(* Logix 5000 project; controller PRU vendor 1 type 14 code 107 rev 20.13; software revision 20.01; part 15 of 17 *)
(* tags used below, declared in another part *)
   AFI : BOOL;
   CMD_LEFT_SCREW_START : BOOL;
   CMD_LEFT_SCREW_STOP : BOOL;
   CMD_RIGHT_SCREW_START : BOOL;
   CMD_RIGHT_SCREW_STOP : BOOL;
   CONTROLLED_STOP : BOOL;
   COOL_FOR_MOTOR_STOP : BOOL;
   DCS_ESTOP_ION : BOOL;
   DRYER : DUAL_SCREW;
   DRYER_AUTO_MODE_PB_ONS : BOOL;
   DRYER_CENTER_STARTUP_MODE : BOOL;
   DRYER_CENTER_TON : TIMER;
   DRYER_MAN_MODE_PB_ONS : BOOL;
   DRYER_MODE_AUTO : BOOL;
   DRYER_MODE_OFF : BOOL;
   DRYER_ONS : BOOL;
   DRYER_SEMIAUTO_MODE_PB_ONS : BOOL;
   DRYER_SHUTDOWN_FAULT_ION : BOOL;
   ENCODER_ERROR : REAL;
   ESR_CONTACT_1_ION : BOOL;
   ESR_CONTACT_2_ION : BOOL;
   ESTOP_PB_IOF : BOOL;   // E-STOP PUSHBUTTON IS PUSHED.
   FAULT : DINT[100];
   FAULT_DRYERL_MSG_TON : TIMER;
   FAULT_DRYERR_MSG_TON : TIMER;
   FAULT_TIMER : TIMER[10000];
   FAULTS_FA1_IOK : BOOL;   // SYSTEM LEVEL FAULTS ARE OK.
   FAULTS_FA1A_IOK : BOOL;   // MODULE FAULTS ARE OK.
   FAULTS_FA1B_IOK : BOOL;   // STOP PUSHBUTTON FAULTS ARE OK.
   FAULTS_FA3A_IOK : BOOL;   // SCREWS DRIVES NOT FAULTED.
   HMI_ALARM_RESET : BOOL;
   HMI_DRYER_AUTO_MODE_PB : BOOL;
   HMI_DRYER_MAN_MODE_PB : BOOL;
   HMI_DRYER_OFF_MODE_PB : BOOL;
   HMI_DRYER_SEMIAUTO_MODE_PB : BOOL;
   HMI_DRYERL_SPEED : REAL;
   HMI_DRYERR_SPEED : REAL;
   HMI_STOP_ALL : BOOL;
   HMI_SYSTEM_AUTO_MODE_PB : BOOL;
   HMI_VFD_1_JOG_FWD_PB : BOOL;
   HMI_VFD_1_JOG_REV_PB : BOOL;
   HMI_VFD_2_JOG_FWD_PB : BOOL;
   HMI_VFD_2_JOG_REV_PB : BOOL;
   MODE_DRYER : INT;
   Module_DRYERL_Fault : DINT;
   Module_DRYERL_Iok : BOOL;
   Module_DRYERL_Status : DINT;
   Module_DRYERR_Fault : DINT;
   Module_DRYERR_Iok : BOOL;
   Module_DRYERR_Status : DINT;
   OK_TO_STOP : BOOL;
   PF70EL_Message : MESSAGE;
   PF70ER_Message : MESSAGE;
   PROCESS_SEQUENCER : INT;
   REQUEST_TO_STOP : BOOL;   // HMI MIXING SCREEN - REQUEST TO STOP WHEN SCREWS ARE NEAR ZERO.
   REQUEST_TO_STOP_L : BOOL;
   SCREWS_ENABLE_GON : BOOL;   // Dryer screw faults are ok.
   THRESHOLD : REAL[9000];
   VFD_1_Current_Real : REAL;
   VFD_2_Current_Real : REAL;
   VFD_CommsFaultTest : DINT;
   VFDS_BON : BOOL;   // DRYER VFDs HAVE BEEN COMMANDED ON FOR 1 SECOND.
   VFDS_TON : TIMER;

PROGRAM SCREW_CONTROL   (* main routine DUALSCREW *)

ROUTINE A01_DRYER_Start_Stop   (* ladder *)
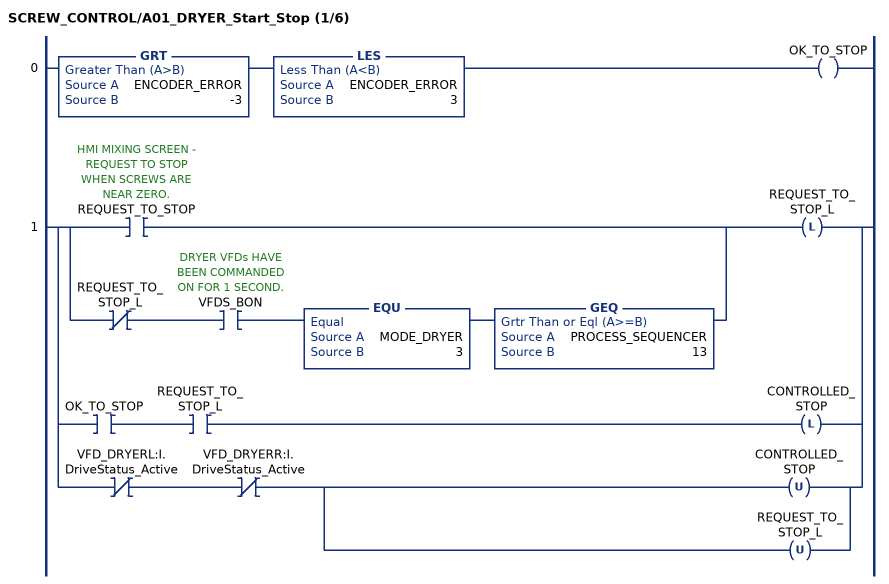
   0: GRT(ENCODER_ERROR,-3)LES(ENCODER_ERROR,3)OTE(OK_TO_STOP);
   1: [[XIC(REQUEST_TO_STOP) ,XIO(REQUEST_TO_STOP_L) XIC(VFDS_BON) EQU(MODE_DRYER,3) GEQ(PROCESS_SEQUENCER,13) ] OTL(REQUEST_TO_STOP_L) ,XIC(OK_TO_STOP) XIC(REQUEST_TO_STOP_L) OTL(CONTROLLED_STOP) ,XIO(VFD_DRYERL:I.DriveStatus_Active) XIO(VFD_DRYERR:I.DriveStatus_Active) [OTU(CONTROLLED_STOP) ,OTU(REQUEST_TO_STOP_L) ] ];
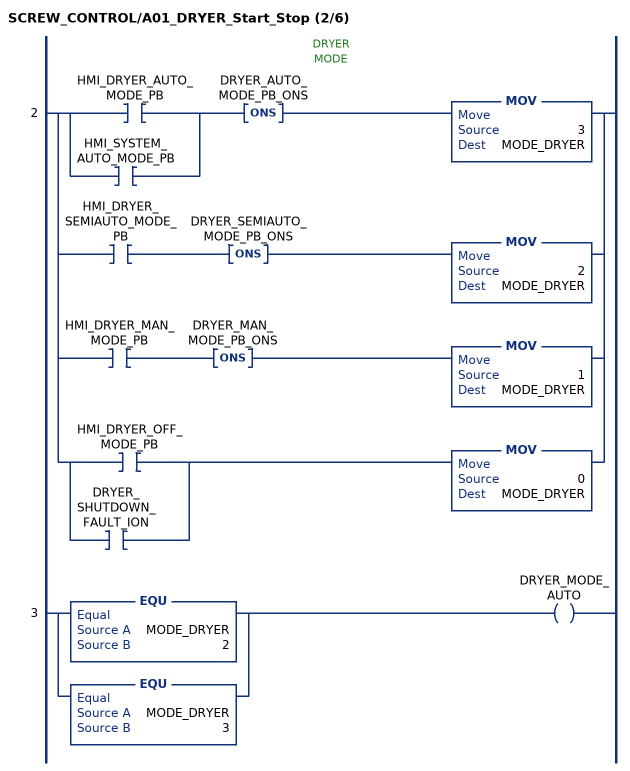
   // DRYER
   // MODE
   2: [[XIC(HMI_DRYER_AUTO_MODE_PB) ,XIC(HMI_SYSTEM_AUTO_MODE_PB) ] ONS(DRYER_AUTO_MODE_PB_ONS) MOV(3,MODE_DRYER) ,XIC(HMI_DRYER_SEMIAUTO_MODE_PB) ONS(DRYER_SEMIAUTO_MODE_PB_ONS) MOV(2,MODE_DRYER) ,XIC(HMI_DRYER_MAN_MODE_PB) ONS(DRYER_MAN_MODE_PB_ONS) MOV(1,MODE_DRYER) ,[XIC(HMI_DRYER_OFF_MODE_PB) ,XIC(DRYER_SHUTDOWN_FAULT_ION) ] MOV(0,MODE_DRYER) ];
   3: [EQU(MODE_DRYER,2) ,EQU(MODE_DRYER,3) ]OTE(DRYER_MODE_AUTO);
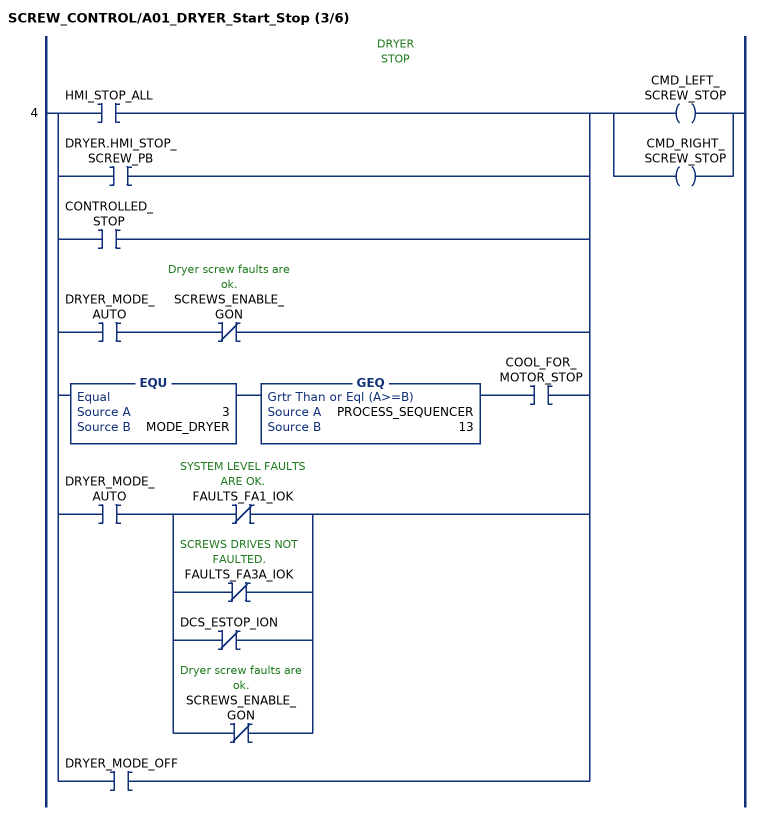
   // DRYER
   // STOP
   4: [XIC(HMI_STOP_ALL) ,XIC(DRYER.HMI_STOP_SCREW_PB) ,XIC(CONTROLLED_STOP) ,XIC(DRYER_MODE_AUTO) XIO(SCREWS_ENABLE_GON) ,EQU(3,MODE_DRYER) GEQ(PROCESS_SEQUENCER,13) XIC(COOL_FOR_MOTOR_STOP) ,XIC(DRYER_MODE_AUTO) [XIO(FAULTS_FA1_IOK) ,XIO(FAULTS_FA3A_IOK) ,XIO(DCS_ESTOP_ION) ,XIO(SCREWS_ENABLE_GON) ] ,XIC(DRYER_MODE_OFF) ][OTE(CMD_LEFT_SCREW_STOP) ,OTE(CMD_RIGHT_SCREW_STOP) ];
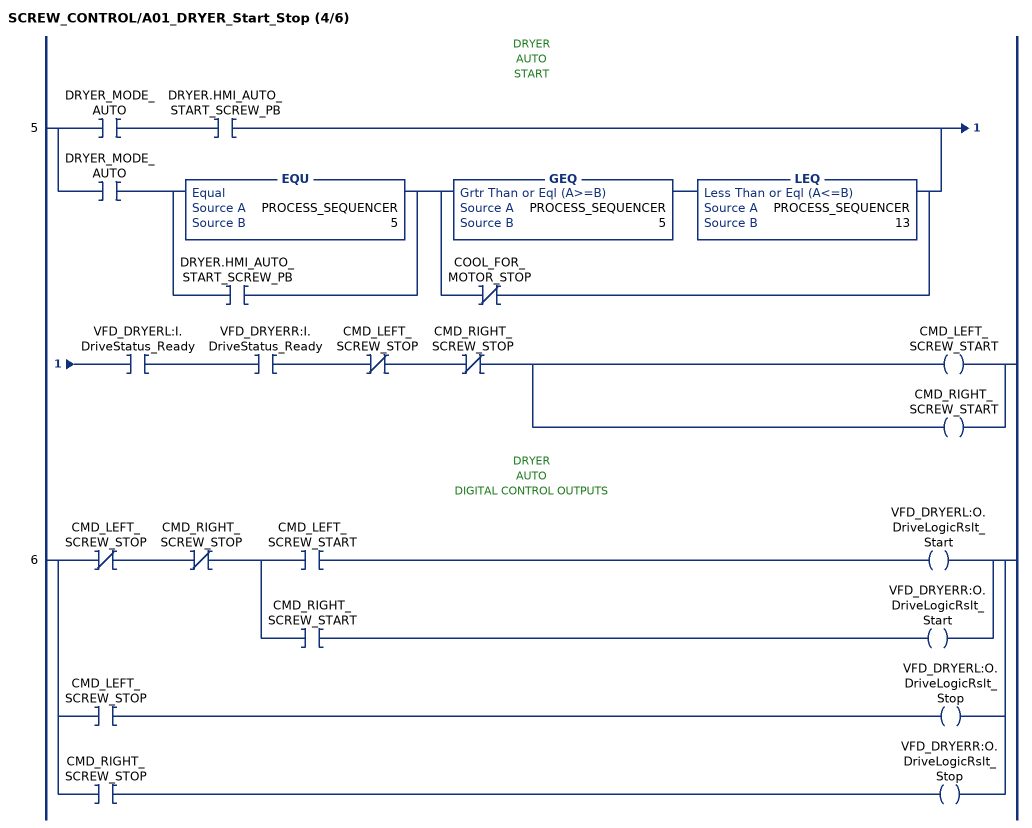
   // DRYER
   // AUTO
   //  START
   5: [XIC(DRYER_MODE_AUTO) XIC(DRYER.HMI_AUTO_START_SCREW_PB) ,XIC(DRYER_MODE_AUTO) [EQU(PROCESS_SEQUENCER,5) ,XIC(DRYER.HMI_AUTO_START_SCREW_PB) ] [GEQ(PROCESS_SEQUENCER,5) LEQ(PROCESS_SEQUENCER,13) ,XIO(COOL_FOR_MOTOR_STOP) ] ]XIC(VFD_DRYERL:I.DriveStatus_Ready)XIC(VFD_DRYERR:I.DriveStatus_Ready)XIO(CMD_LEFT_SCREW_STOP)XIO(CMD_RIGHT_SCREW_STOP)[OTE(CMD_LEFT_SCREW_START) ,OTE(CMD_RIGHT_SCREW_START) ];
   // DRYER
   // AUTO
   // DIGITAL CONTROL OUTPUTS
   6: [XIO(CMD_LEFT_SCREW_STOP) XIO(CMD_RIGHT_SCREW_STOP) [XIC(CMD_LEFT_SCREW_START) OTE(VFD_DRYERL:O.DriveLogicRslt_Start) ,XIC(CMD_RIGHT_SCREW_START) OTE(VFD_DRYERR:O.DriveLogicRslt_Start) ] ,XIC(CMD_LEFT_SCREW_STOP) OTE(VFD_DRYERL:O.DriveLogicRslt_Stop) ,XIC(CMD_RIGHT_SCREW_STOP) OTE(VFD_DRYERR:O.DriveLogicRslt_Stop) ];
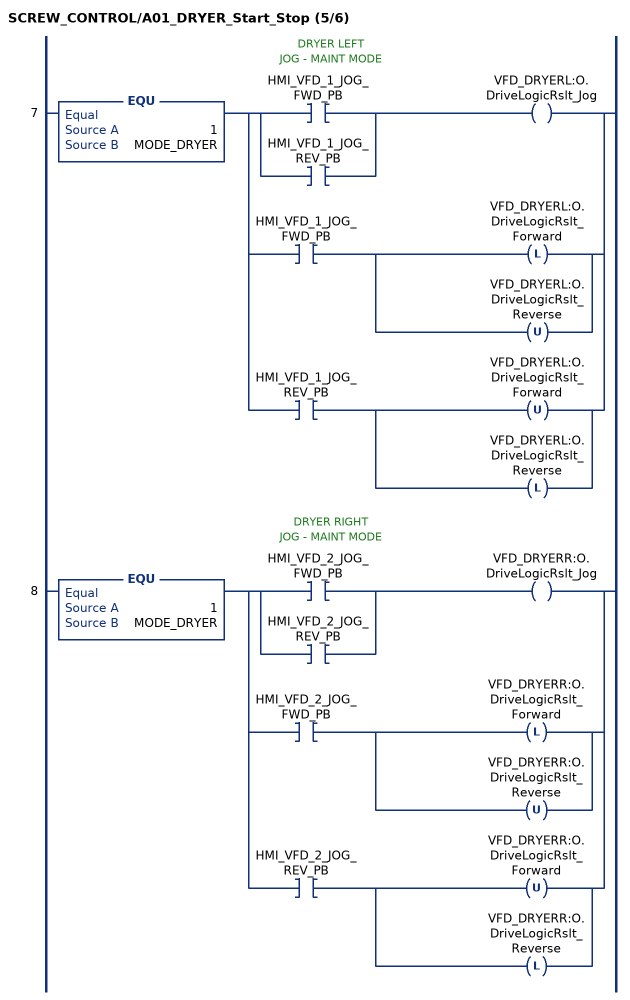
   // DRYER LEFT
   // JOG - MAINT MODE
   7: EQU(1,MODE_DRYER)[[XIC(HMI_VFD_1_JOG_FWD_PB) ,XIC(HMI_VFD_1_JOG_REV_PB) ] OTE(VFD_DRYERL:O.DriveLogicRslt_Jog) ,XIC(HMI_VFD_1_JOG_FWD_PB) [OTL(VFD_DRYERL:O.DriveLogicRslt_Forward) ,OTU(VFD_DRYERL:O.DriveLogicRslt_Reverse) ] ,XIC(HMI_VFD_1_JOG_REV_PB) [OTU(VFD_DRYERL:O.DriveLogicRslt_Forward) ,OTL(VFD_DRYERL:O.DriveLogicRslt_Reverse) ] ];
   // DRYER RIGHT
   // JOG - MAINT MODE
   8: EQU(1,MODE_DRYER)[[XIC(HMI_VFD_2_JOG_FWD_PB) ,XIC(HMI_VFD_2_JOG_REV_PB) ] OTE(VFD_DRYERR:O.DriveLogicRslt_Jog) ,XIC(HMI_VFD_2_JOG_FWD_PB) [OTL(VFD_DRYERR:O.DriveLogicRslt_Forward) ,OTU(VFD_DRYERR:O.DriveLogicRslt_Reverse) ] ,XIC(HMI_VFD_2_JOG_REV_PB) [OTU(VFD_DRYERR:O.DriveLogicRslt_Forward) ,OTL(VFD_DRYERR:O.DriveLogicRslt_Reverse) ] ];
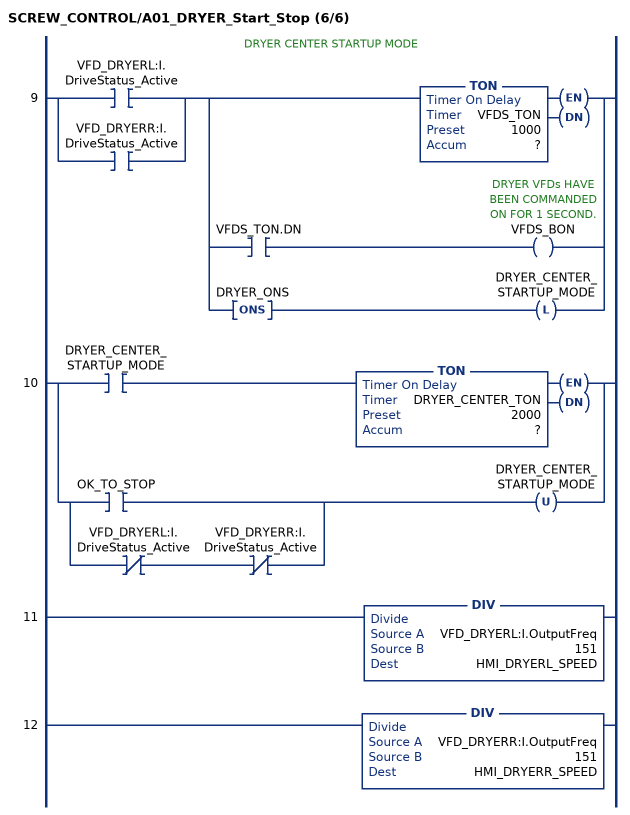
   // DRYER CENTER STARTUP MODE
   9: [XIC(VFD_DRYERL:I.DriveStatus_Active) ,XIC(VFD_DRYERR:I.DriveStatus_Active) ][TON(VFDS_TON,?,?) ,XIC(VFDS_TON.DN) OTE(VFDS_BON) ,ONS(DRYER_ONS) OTL(DRYER_CENTER_STARTUP_MODE) ];
   10: [XIC(DRYER_CENTER_STARTUP_MODE) TON(DRYER_CENTER_TON,?,?) ,[XIC(OK_TO_STOP) ,XIO(VFD_DRYERL:I.DriveStatus_Active) XIO(VFD_DRYERR:I.DriveStatus_Active) ] OTU(DRYER_CENTER_STARTUP_MODE) ];
   11: DIV(VFD_DRYERL:I.OutputFreq,151,HMI_DRYERL_SPEED);
   12: DIV(VFD_DRYERR:I.OutputFreq,151,HMI_DRYERR_SPEED);
END_ROUTINE

ROUTINE B01_FA1_B_FAULTS_1200_STOP   (* ladder *)
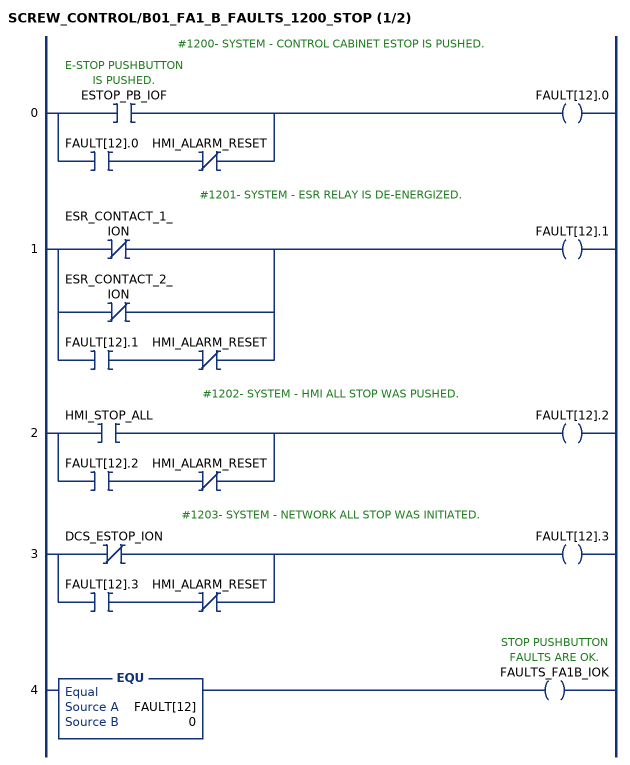
   // #1200- SYSTEM - CONTROL CABINET ESTOP IS PUSHED.
   0: [XIC(ESTOP_PB_IOF) ,XIC(FAULT[12].0) XIO(HMI_ALARM_RESET) ]OTE(FAULT[12].0);
   // #1201- SYSTEM - ESR RELAY IS DE-ENERGIZED.
   1: [XIO(ESR_CONTACT_1_ION) ,XIO(ESR_CONTACT_2_ION) ,XIC(FAULT[12].1) XIO(HMI_ALARM_RESET) ]OTE(FAULT[12].1);
   // #1202- SYSTEM - HMI ALL STOP WAS PUSHED.
   2: [XIC(HMI_STOP_ALL) ,XIC(FAULT[12].2) XIO(HMI_ALARM_RESET) ]OTE(FAULT[12].2);
   // #1203- SYSTEM - NETWORK ALL STOP WAS INITIATED.
   3: [XIO(DCS_ESTOP_ION) ,XIC(FAULT[12].3) XIO(HMI_ALARM_RESET) ]OTE(FAULT[12].3);
   4: EQU(FAULT[12],0)OTE(FAULTS_FA1B_IOK);
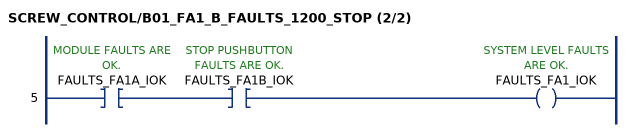
   5: XIC(FAULTS_FA1A_IOK)XIC(FAULTS_FA1B_IOK)OTE(FAULTS_FA1_IOK);
END_ROUTINE

ROUTINE B03_FA3_A_PYROSCREW_FAULTS_3000   (* ladder *)
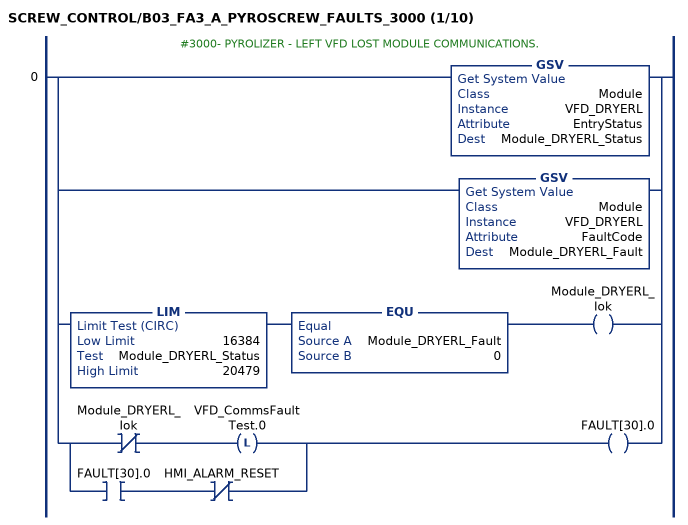
   // #3000- PYROLIZER - LEFT VFD LOST MODULE COMMUNICATIONS.
   0: [GSV(Module,VFD_DRYERL,EntryStatus,Module_DRYERL_Status) ,GSV(Module,VFD_DRYERL,FaultCode,Module_DRYERL_Fault) ,LIM(16384,Module_DRYERL_Status,20479) EQU(Module_DRYERL_Fault,0) OTE(Module_DRYERL_Iok) ,[XIO(Module_DRYERL_Iok) OTL(VFD_CommsFaultTest.0) ,XIC(FAULT[30].0) XIO(HMI_ALARM_RESET) ] OTE(FAULT[30].0) ];
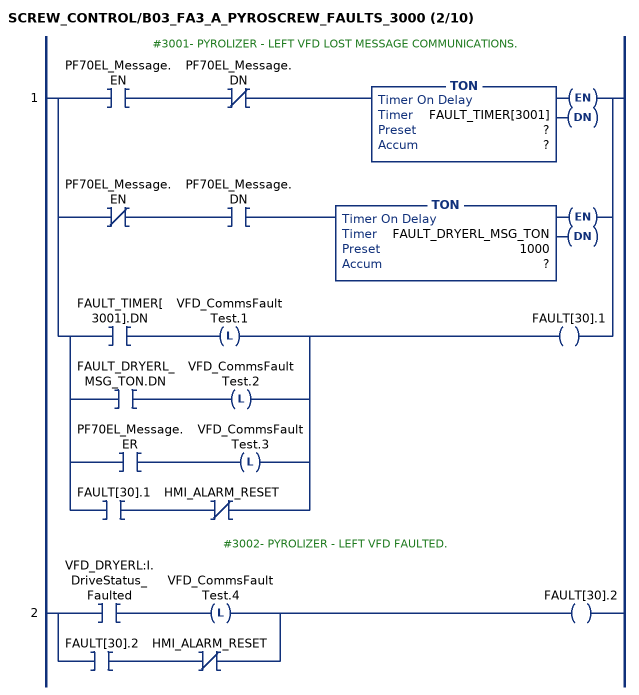
   // #3001- PYROLIZER - LEFT VFD LOST MESSAGE COMMUNICATIONS.
   1: [XIC(PF70EL_Message.EN) XIO(PF70EL_Message.DN) TON(FAULT_TIMER[3001],?,?) ,XIO(PF70EL_Message.EN) XIC(PF70EL_Message.DN) TON(FAULT_DRYERL_MSG_TON,?,?) ,[XIC(FAULT_TIMER[3001].DN) OTL(VFD_CommsFaultTest.1) ,XIC(FAULT_DRYERL_MSG_TON.DN) OTL(VFD_CommsFaultTest.2) ,XIC(PF70EL_Message.ER) OTL(VFD_CommsFaultTest.3) ,XIC(FAULT[30].1) XIO(HMI_ALARM_RESET) ] OTE(FAULT[30].1) ];
   // #3002- PYROLIZER - LEFT VFD FAULTED.
   2: [XIC(VFD_DRYERL:I.DriveStatus_Faulted) OTL(VFD_CommsFaultTest.4) ,XIC(FAULT[30].2) XIO(HMI_ALARM_RESET) ]OTE(FAULT[30].2);
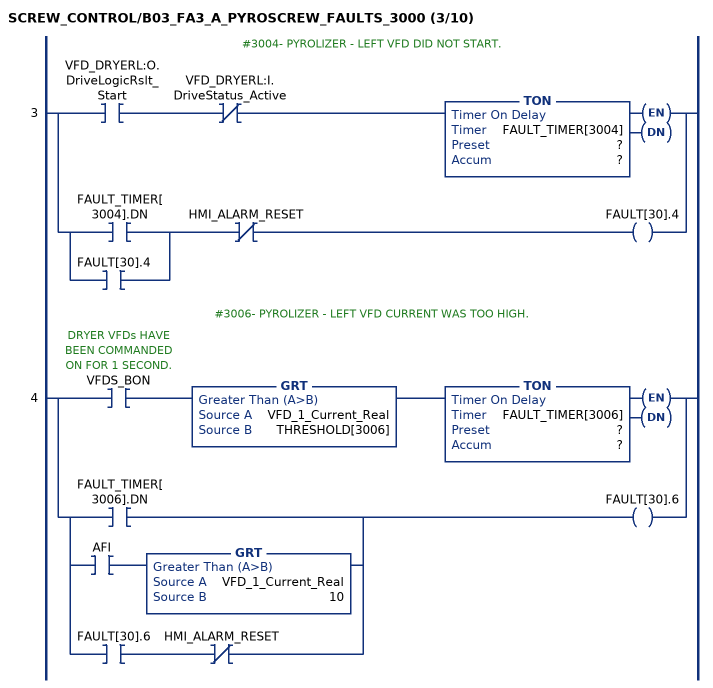
   // #3004- PYROLIZER - LEFT VFD DID NOT START.
   3: [XIC(VFD_DRYERL:O.DriveLogicRslt_Start) XIO(VFD_DRYERL:I.DriveStatus_Active) TON(FAULT_TIMER[3004],?,?) ,[XIC(FAULT_TIMER[3004].DN) ,XIC(FAULT[30].4) ] XIO(HMI_ALARM_RESET) OTE(FAULT[30].4) ];
   // #3006- PYROLIZER - LEFT VFD CURRENT WAS TOO HIGH.
   4: [XIC(VFDS_BON) GRT(VFD_1_Current_Real,THRESHOLD[3006]) TON(FAULT_TIMER[3006],?,?) ,[XIC(FAULT_TIMER[3006].DN) ,XIC(AFI) GRT(VFD_1_Current_Real,10) ,XIC(FAULT[30].6) XIO(HMI_ALARM_RESET) ] OTE(FAULT[30].6) ];
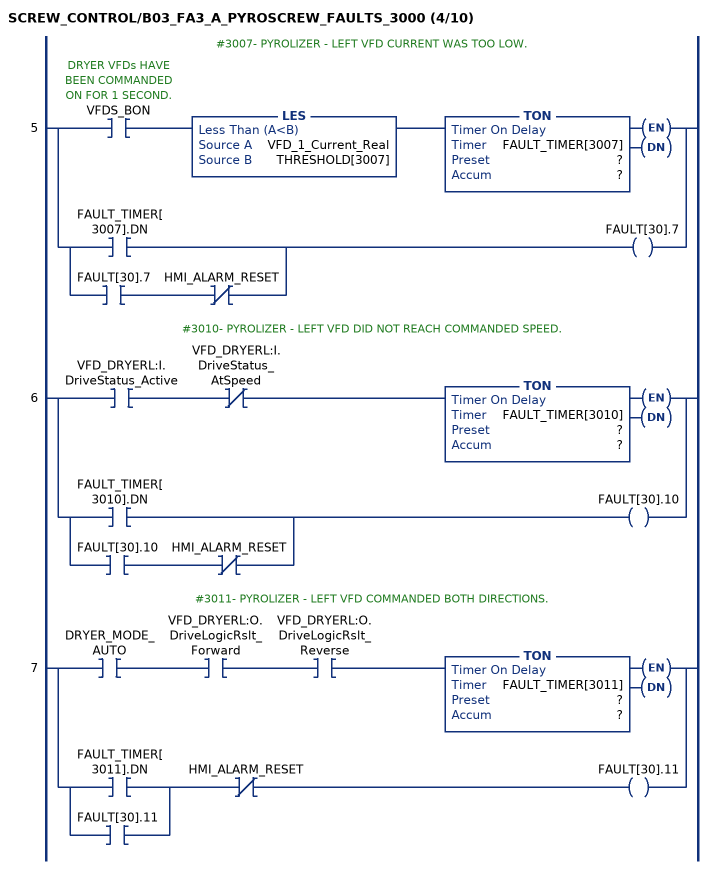
   // #3007- PYROLIZER - LEFT VFD CURRENT WAS TOO LOW.
   5: [XIC(VFDS_BON) LES(VFD_1_Current_Real,THRESHOLD[3007]) TON(FAULT_TIMER[3007],?,?) ,[XIC(FAULT_TIMER[3007].DN) ,XIC(FAULT[30].7) XIO(HMI_ALARM_RESET) ] OTE(FAULT[30].7) ];
   // #3010- PYROLIZER - LEFT VFD DID NOT REACH COMMANDED SPEED.
   6: [XIC(VFD_DRYERL:I.DriveStatus_Active) XIO(VFD_DRYERL:I.DriveStatus_AtSpeed) TON(FAULT_TIMER[3010],?,?) ,[XIC(FAULT_TIMER[3010].DN) ,XIC(FAULT[30].10) XIO(HMI_ALARM_RESET) ] OTE(FAULT[30].10) ];
   // #3011- PYROLIZER - LEFT VFD COMMANDED BOTH DIRECTIONS.
   7: [XIC(DRYER_MODE_AUTO) XIC(VFD_DRYERL:O.DriveLogicRslt_Forward) XIC(VFD_DRYERL:O.DriveLogicRslt_Reverse) TON(FAULT_TIMER[3011],?,?) ,[XIC(FAULT_TIMER[3011].DN) ,XIC(FAULT[30].11) ] XIO(HMI_ALARM_RESET) OTE(FAULT[30].11) ];
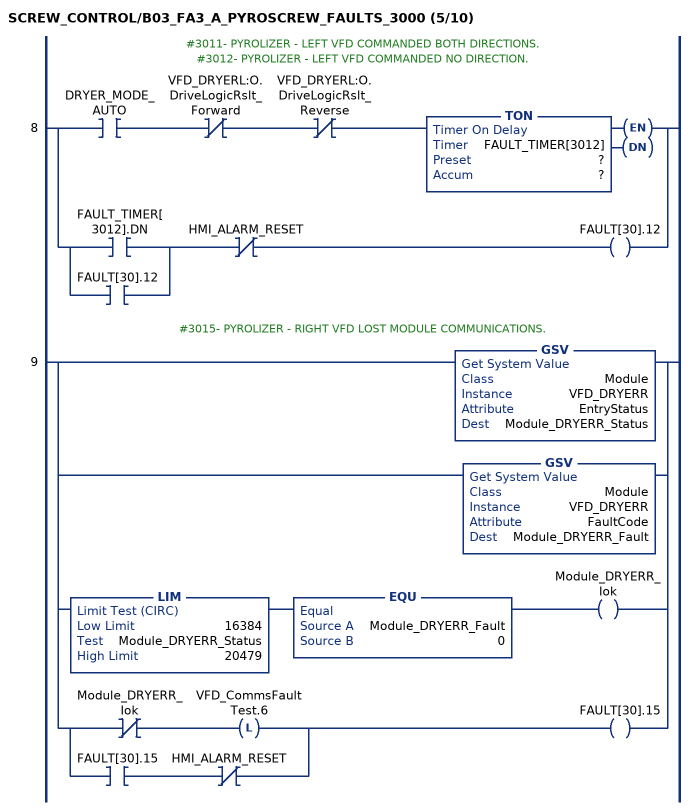
   // #3011- PYROLIZER - LEFT VFD COMMANDED BOTH DIRECTIONS.
   // #3012- PYROLIZER - LEFT VFD COMMANDED NO DIRECTION.
   8: [XIC(DRYER_MODE_AUTO) XIO(VFD_DRYERL:O.DriveLogicRslt_Forward) XIO(VFD_DRYERL:O.DriveLogicRslt_Reverse) TON(FAULT_TIMER[3012],?,?) ,[XIC(FAULT_TIMER[3012].DN) ,XIC(FAULT[30].12) ] XIO(HMI_ALARM_RESET) OTE(FAULT[30].12) ];
   // #3015- PYROLIZER - RIGHT VFD LOST MODULE COMMUNICATIONS.
   9: [GSV(Module,VFD_DRYERR,EntryStatus,Module_DRYERR_Status) ,GSV(Module,VFD_DRYERR,FaultCode,Module_DRYERR_Fault) ,LIM(16384,Module_DRYERR_Status,20479) EQU(Module_DRYERR_Fault,0) OTE(Module_DRYERR_Iok) ,[XIO(Module_DRYERR_Iok) OTL(VFD_CommsFaultTest.6) ,XIC(FAULT[30].15) XIO(HMI_ALARM_RESET) ] OTE(FAULT[30].15) ];
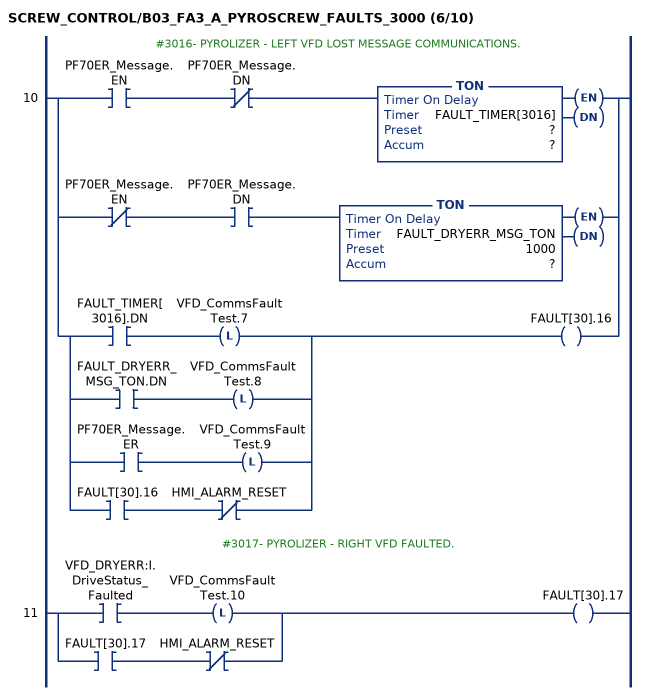
   // #3016- PYROLIZER - LEFT VFD LOST MESSAGE COMMUNICATIONS.
   10: [XIC(PF70ER_Message.EN) XIO(PF70ER_Message.DN) TON(FAULT_TIMER[3016],?,?) ,XIO(PF70ER_Message.EN) XIC(PF70ER_Message.DN) TON(FAULT_DRYERR_MSG_TON,?,?) ,[XIC(FAULT_TIMER[3016].DN) OTL(VFD_CommsFaultTest.7) ,XIC(FAULT_DRYERR_MSG_TON.DN) OTL(VFD_CommsFaultTest.8) ,XIC(PF70ER_Message.ER) OTL(VFD_CommsFaultTest.9) ,XIC(FAULT[30].16) XIO(HMI_ALARM_RESET) ] OTE(FAULT[30].16) ];
   // #3017- PYROLIZER - RIGHT VFD FAULTED.
   11: [XIC(VFD_DRYERR:I.DriveStatus_Faulted) OTL(VFD_CommsFaultTest.10) ,XIC(FAULT[30].17) XIO(HMI_ALARM_RESET) ]OTE(FAULT[30].17);
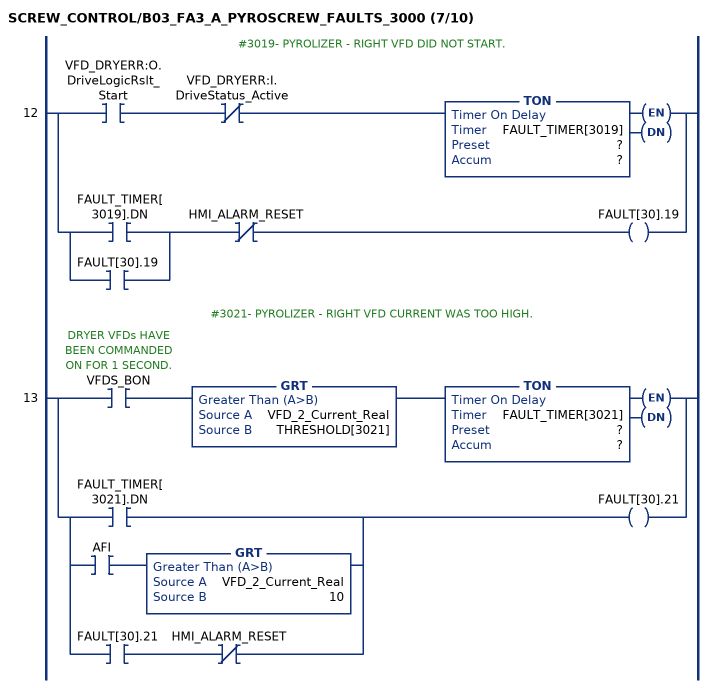
   // #3019- PYROLIZER - RIGHT VFD DID NOT START.
   12: [XIC(VFD_DRYERR:O.DriveLogicRslt_Start) XIO(VFD_DRYERR:I.DriveStatus_Active) TON(FAULT_TIMER[3019],?,?) ,[XIC(FAULT_TIMER[3019].DN) ,XIC(FAULT[30].19) ] XIO(HMI_ALARM_RESET) OTE(FAULT[30].19) ];
   // #3021- PYROLIZER - RIGHT VFD CURRENT WAS TOO HIGH.
   13: [XIC(VFDS_BON) GRT(VFD_2_Current_Real,THRESHOLD[3021]) TON(FAULT_TIMER[3021],?,?) ,[XIC(FAULT_TIMER[3021].DN) ,XIC(AFI) GRT(VFD_2_Current_Real,10) ,XIC(FAULT[30].21) XIO(HMI_ALARM_RESET) ] OTE(FAULT[30].21) ];
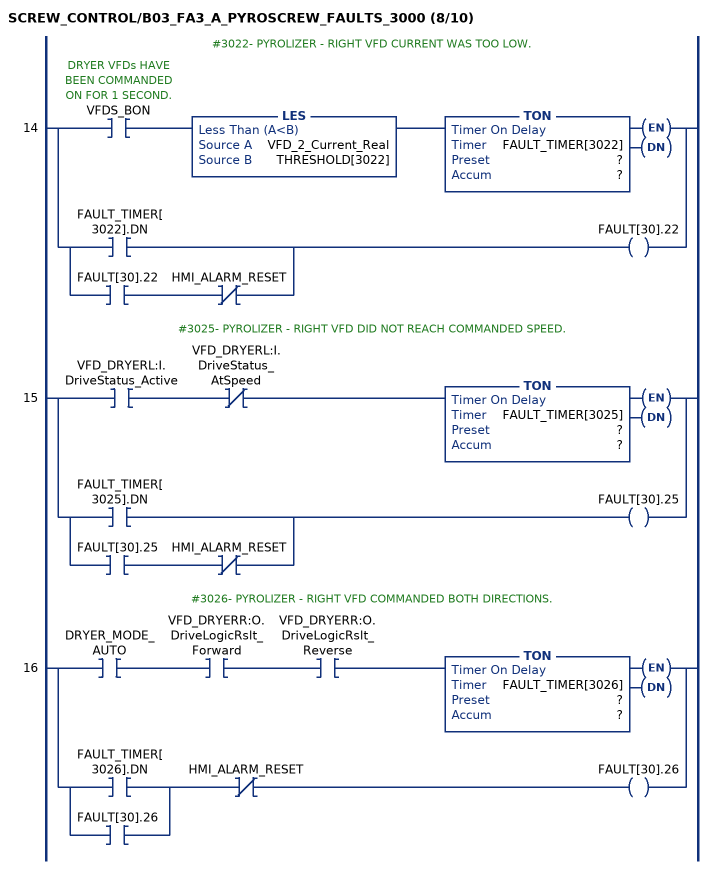
   // #3022- PYROLIZER - RIGHT VFD CURRENT WAS TOO LOW.
   14: [XIC(VFDS_BON) LES(VFD_2_Current_Real,THRESHOLD[3022]) TON(FAULT_TIMER[3022],?,?) ,[XIC(FAULT_TIMER[3022].DN) ,XIC(FAULT[30].22) XIO(HMI_ALARM_RESET) ] OTE(FAULT[30].22) ];
   // #3025- PYROLIZER - RIGHT VFD DID NOT REACH COMMANDED SPEED.
   15: [XIC(VFD_DRYERL:I.DriveStatus_Active) XIO(VFD_DRYERL:I.DriveStatus_AtSpeed) TON(FAULT_TIMER[3025],?,?) ,[XIC(FAULT_TIMER[3025].DN) ,XIC(FAULT[30].25) XIO(HMI_ALARM_RESET) ] OTE(FAULT[30].25) ];
   // #3026- PYROLIZER - RIGHT VFD COMMANDED BOTH DIRECTIONS.
   16: [XIC(DRYER_MODE_AUTO) XIC(VFD_DRYERR:O.DriveLogicRslt_Forward) XIC(VFD_DRYERR:O.DriveLogicRslt_Reverse) TON(FAULT_TIMER[3026],?,?) ,[XIC(FAULT_TIMER[3026].DN) ,XIC(FAULT[30].26) ] XIO(HMI_ALARM_RESET) OTE(FAULT[30].26) ];
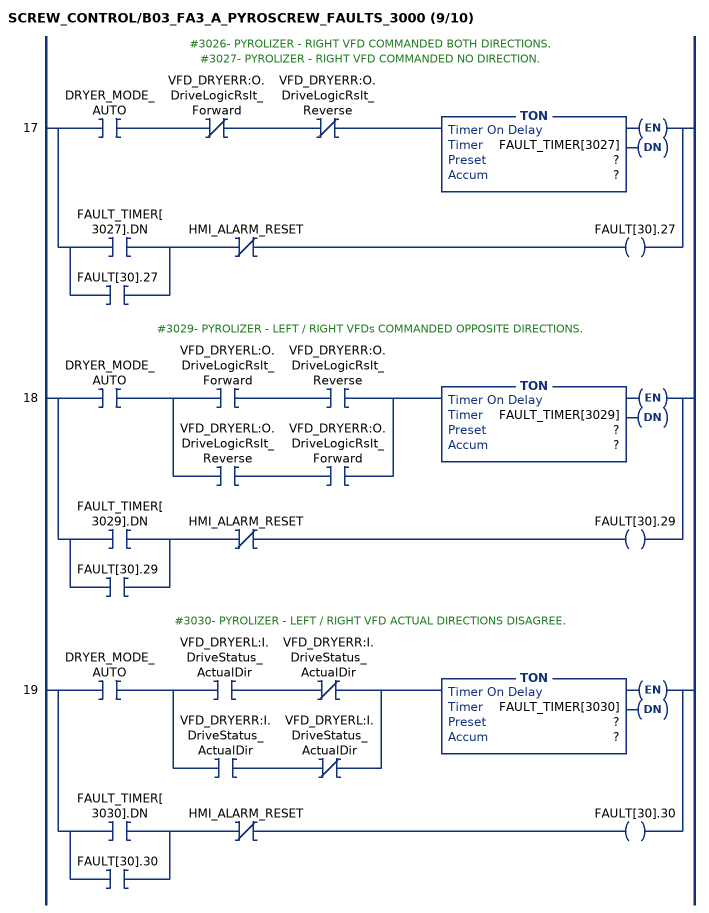
   // #3026- PYROLIZER - RIGHT VFD COMMANDED BOTH DIRECTIONS.
   // #3027- PYROLIZER - RIGHT VFD COMMANDED NO DIRECTION.
   17: [XIC(DRYER_MODE_AUTO) XIO(VFD_DRYERR:O.DriveLogicRslt_Forward) XIO(VFD_DRYERR:O.DriveLogicRslt_Reverse) TON(FAULT_TIMER[3027],?,?) ,[XIC(FAULT_TIMER[3027].DN) ,XIC(FAULT[30].27) ] XIO(HMI_ALARM_RESET) OTE(FAULT[30].27) ];
   // #3029- PYROLIZER - LEFT / RIGHT VFDs COMMANDED OPPOSITE DIRECTIONS.
   18: [XIC(DRYER_MODE_AUTO) [XIC(VFD_DRYERL:O.DriveLogicRslt_Forward) XIC(VFD_DRYERR:O.DriveLogicRslt_Reverse) ,XIC(VFD_DRYERL:O.DriveLogicRslt_Reverse) XIC(VFD_DRYERR:O.DriveLogicRslt_Forward) ] TON(FAULT_TIMER[3029],?,?) ,[XIC(FAULT_TIMER[3029].DN) ,XIC(FAULT[30].29) ] XIO(HMI_ALARM_RESET) OTE(FAULT[30].29) ];
   // #3030- PYROLIZER - LEFT / RIGHT VFD ACTUAL DIRECTIONS DISAGREE.
   19: [XIC(DRYER_MODE_AUTO) [XIC(VFD_DRYERL:I.DriveStatus_ActualDir) XIO(VFD_DRYERR:I.DriveStatus_ActualDir) ,XIC(VFD_DRYERR:I.DriveStatus_ActualDir) XIO(VFD_DRYERL:I.DriveStatus_ActualDir) ] TON(FAULT_TIMER[3030],?,?) ,[XIC(FAULT_TIMER[3030].DN) ,XIC(FAULT[30].30) ] XIO(HMI_ALARM_RESET) OTE(FAULT[30].30) ];
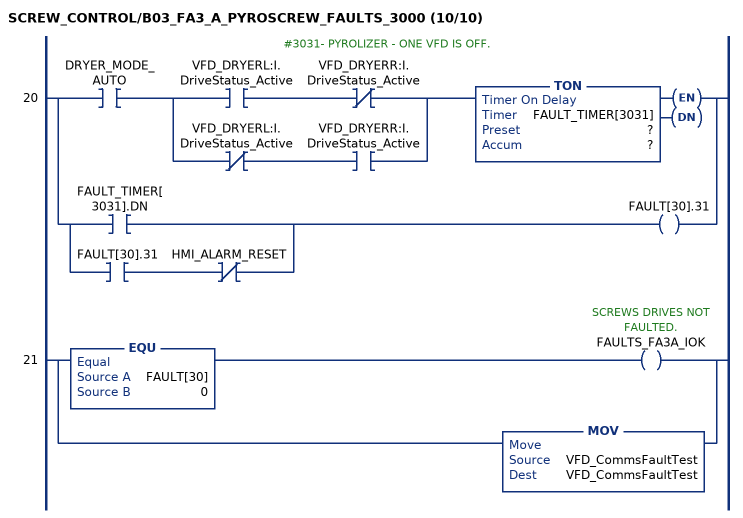
   // #3031- PYROLIZER - ONE VFD IS OFF.
   20: [XIC(DRYER_MODE_AUTO) [XIC(VFD_DRYERL:I.DriveStatus_Active) XIO(VFD_DRYERR:I.DriveStatus_Active) ,XIO(VFD_DRYERL:I.DriveStatus_Active) XIC(VFD_DRYERR:I.DriveStatus_Active) ] TON(FAULT_TIMER[3031],?,?) ,[XIC(FAULT_TIMER[3031].DN) ,XIC(FAULT[30].31) XIO(HMI_ALARM_RESET) ] OTE(FAULT[30].31) ];
   21: [EQU(FAULT[30],0) OTE(FAULTS_FA3A_IOK) ,MOV(VFD_CommsFaultTest,VFD_CommsFaultTest) ];
END_ROUTINE
